TYPE MicroEpsilonDistanceSensorConfig EXTENDS DeviceConfiguration :
STRUCT
END_STRUCT
END_TYPE

(* stored: Version 1.1.0.1, ProductVersion 3.1.4024.12
   DUT MicroEpsilonDistanceSensorConfig: Id {e5f64eb5-da8c-4fe7-8f43-a8c32fb93748} *)
